FUNCTION_BLOCK fbMainStationProcess

VAR_INPUT
	(*fbStnSeqProcess*)
	bSavePB_Uni 									: BOOL; 														(*Universal*) (* Input - HMI - Save Push Button on Touchscreen*)
	bLoadPB_Uni 								: BOOL;														(*Universal*) (* Input - HMI - Load Push Button on Touchscreen*)
	bTrackerEn									: BOOL;														(*During Tracker, it will only call arm when process completed*)
	bTrackerBasedOnPreviousTime			: BOOL;

	(*fbGnrStationMasterController*)
	iCurrentStationAddress_Fix 					: INT;															(*Individual*) (* Input - Define current station no so that this fb know which array number to used*)
	iPreCallArmTime_Uni						: INT;															(*Universal*) (* Input - Pre-Call Arm Time, Program will call arm if the Total process timeEV Equal or Lesser than this value*)
	ARbAlternateStnEn : ARRAY [1..iAlternateSetQty] OF BOOL;
	AR2siAlternateStn : ARRAY [1..iAlternateSetQty, 1..iAlternateStnQty] OF INT;


END_VAR

VAR_IN_OUT PERSISTENT

	(*fbStnSeqProcess*)
(*	DsStnSeqProInput_Ind 						: DS_StnSeqProInput;											(*Individual*) (* Input - PV of Instrument (Temperature, pressure, vacuum and etc), Signal of Sensor to allowed program under the current station status.*)
*)	DSStnSeqProcessCtrl_Ind			 		: DS_fbStnSeqProcessCtrl;									(*Individual*) (* InOut - Link with fbStnSeqProcess, so that this fb know the full status of fbStnSeqProcess and determine which action to take*)

	DsStnSeqRepStore_Ind 						: DS_fbStationSequenceRecipeStore; 						(*Individual*) (* InOut - HMI - The full set of DataStructure-StationSequenceRecipe should selectively display on HMI so that user can customise the recipe by choosing/configure the parameters.*)
	DsStnSubRepStore_Ind 						: DS_fbStationSubRecipeStore; 								(*Individual*) (* InOut - HMI - The full set of DataStructure-StationSubRecipe should selectively display on HMI so that user can customise the recipe by choosing/configure the parameters.*)
	DsStnSeqRepCall_Ind 						: DS_fbStationSequenceRecipeCall;							(*Individual*) (* InOut - Used to call StationSequenceRecipe Detail from fbStationSequenceRecipe*)
	DsStnSubRepCall_Ind 						: DS_fbStationSubRecipeCall;								(*Individual*) (* InOut - Used to call StationSubRecipe Detail from fbStationSubRecipe*)

	(*fbGnrStationMasterController*)
	ARbProductRecipeCallEn_Uni 				: ARRAY [0..iStnQty] OF BOOL;					(*Universal*) (* Output - Link with fbGnrProductRecipeMemory, Array based on Current Station No, the fbGnrProductRecipeMemory will start Read info from Memory when this bool turn on*)
	ARiProductRecipeNoCall_Uni 				: ARRAY [0..iStnQty] OF INT;						(*Universal*) (* Output - Link with fbGnrProductRecipeMemory, Array based on Current Station No, the read out from fbGnrProductRecipeMemory is based on this Product Recipe No*)
	ARiProductRecipeStepCall_Uni 				: ARRAY [0..iStnQty] OF INT;						(*Universal*) (* Output - Link with fbGnrProductRecipeMemory, Array based on Current Station No, the read out from fbGnrProductRecipeMemory is based on this Product Recipe Step No*)

	DSfbGnrProductRecipeMemoryOut_Uni 		: DS_fbGnrProductRecipeMemoryOut;						(*Universal*) (* Input - Link with fbGnrProductRecipeMemory, all the read out info from fbGnrProductRecipeMemory will store in this DataStucture*)

	ARbArmReady_Uni							: ARRAY [1..iArmQty] OF BOOL;								(* Universal*) (* Input  - From ArmPnpFB, This signal is used to confirm if the arm is ready and idling*)

	ARiStnNoToCalledArm_Uni					: ARRAY [0..iArmQty] OF INT; 									(*Universal*) (* Output - Link with fbArmPnP, Array based on Arm No, The Int will store which Station that calling the Arm*)
	ARDSGnrFeedArmPnpParameter_Uni		: ARRAY [0..iArmQty] OF DSGnr_CalledArmPnpParameter; 	(*Universal*) (* Output - Link with fbArmPnP, Array based on Current Station No, Arm should move based on this DataStructure Info*)

	DSLdBasketInfo_Uni		 				: DS_BasketInfo;											(*Input - Loading CONFIRM Basket Info*)
	DSUldBasketInfo_Uni		 				: DS_BasketInfo;											(*Input - Uloading CONFIRM Basket Info*)
	ARDsStnBasketInfo_Uni					: ARRAY [1..iStnQty] OF DS_BasketInfo;						(*Input - Station Basket Info*)



END_VAR

VAR_OUTPUT PERSISTENT
	bSaveInd_Uni 								: BOOL; 														(*Universal*) (* Output - HMI - Save Indicator on Touchscreen*)
	bLoadInd_Uni 								: BOOL; 														(*Universal*) (* Output - HMI - Load Indicator on Touchscreen*)
(*	DSStnSeqProOutput_Ind 						:DS_StnSeqProOutput;										(*Individual*) (* Output - To Control Output - When process running, instrument should control by the output in this Data structure*)
*)
END_VAR



VAR PERSISTENT
	(*fbStnSeqProcess*)
	StnSeqProcessfb: fbStnSeqProcess;
	bStnSeqProcessStartInterlock			: BOOL;															(*Individual*) (* Input - Interlocking to Enable the StnSeqProcess Start Signal, It might used on those station with Sliding door for close confirmation before process start*)

	(*fbGnrStationMasterController*)
	GnrStationMasterControllerfb				: fbGnrStationMasterController;
	bStnSeqProcessSt						: BOOL;															(* Output - Link with fbStnSeqProcess, After Read out from fbGnrProductRecipeMemory, this fb will trigger this Bool to start the StnSeqProcess*)
	DSGnrBufferCalledArmPnpParameter 	: DSGnr_CalledArmPnpParameter;								(* Internal used, Buffer Data Structure read out from fbGnrProductRecipeMemory*)
	DSGnrBuffersPnpSequenceDescription	: STRING (99);														(* Internal used, Buffer Description read out from fbGnrProductRecipeMemory*)
	ARiPreviousStnSeqTotalProcessTime 	: ARRAY [0..iProductRecipeArrayQty] OF INT;					(* Internal used, Previous Total Process Time will save into this Array, Array based on StationSequenceNo*)
	iCallStep									: INT;																(* Internal used, to monitor the current Step so that you can indentify the error of this function block if stucked*)
	DSBasketInfo_Ind 							: DS_BasketInfo;												(*Individual*) (* InOut - Basket Information that comes into current station*)

END_VAR
VAR
	bLdStnConfirm: BOOL;
	bUldStnConfirm: BOOL;
	bStn1Confirm: BOOL;
	bGreaterStn1Confirm: BOOL;
	bLesserStnQtyConfirm: BOOL;
	bEqualStnQtyConfirm: BOOL;
	iTotalProcessTimeSV: INT;
END_VAR
VAR // added by the converter: edge detectors and wires of the graphical bodies
    _w1, _w2, _w3 : DS_BasketInfo;
END_VAR

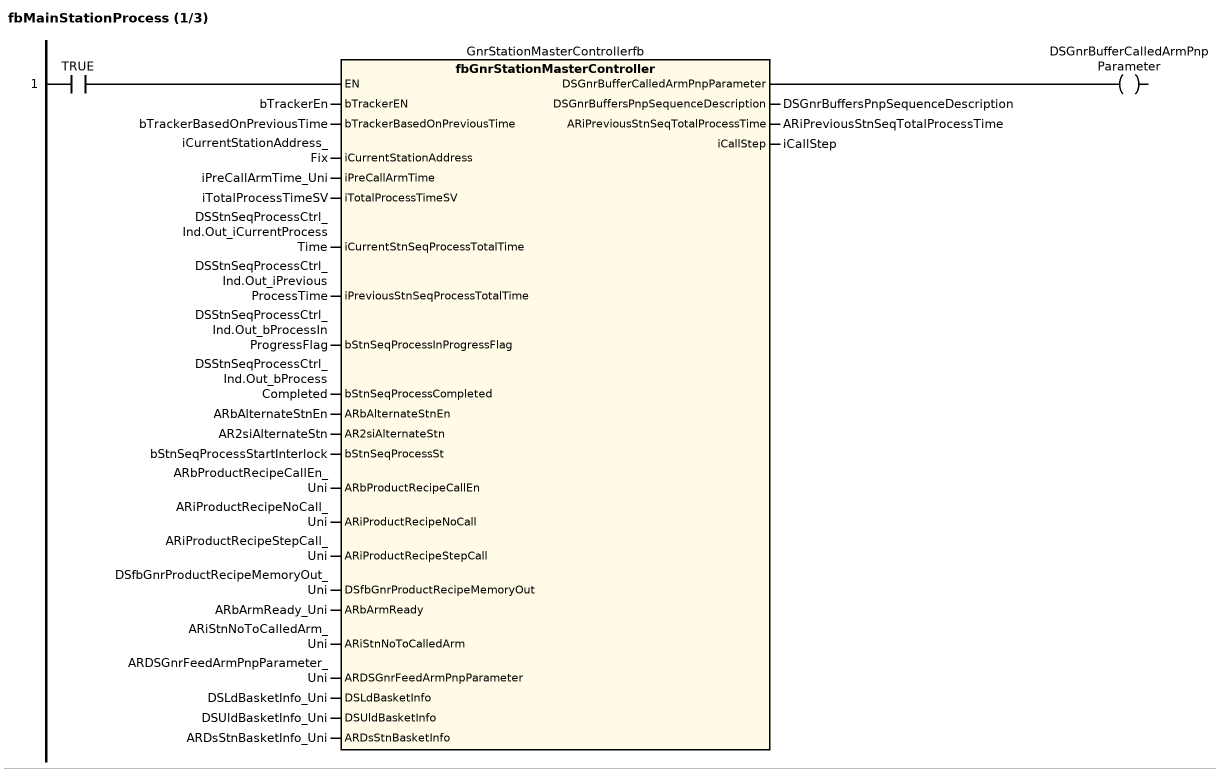
// NETWORK 1
GnrStationMasterControllerfb(
    bTrackerEN := bTrackerEn,
    bTrackerBasedOnPreviousTime := bTrackerBasedOnPreviousTime,
    iCurrentStationAddress := iCurrentStationAddress_Fix,
    iPreCallArmTime := iPreCallArmTime_Uni,
    iTotalProcessTimeSV := iTotalProcessTimeSV,
    iCurrentStnSeqProcessTotalTime := DSStnSeqProcessCtrl_Ind.Out_iCurrentProcessTime,
    iPreviousStnSeqProcessTotalTime := DSStnSeqProcessCtrl_Ind.Out_iPreviousProcessTime,
    bStnSeqProcessInProgressFlag := DSStnSeqProcessCtrl_Ind.Out_bProcessInProgressFlag,
    bStnSeqProcessCompleted := DSStnSeqProcessCtrl_Ind.Out_bProcessCompleted,
    ARbAlternateStnEn := ARbAlternateStnEn,
    AR2siAlternateStn := AR2siAlternateStn,
    bStnSeqProcessSt := bStnSeqProcessStartInterlock,
    ARbProductRecipeCallEn := ARbProductRecipeCallEn_Uni,
    ARiProductRecipeNoCall := ARiProductRecipeNoCall_Uni,
    ARiProductRecipeStepCall := ARiProductRecipeStepCall_Uni,
    DSfbGnrProductRecipeMemoryOut := DSfbGnrProductRecipeMemoryOut_Uni,
    ARbArmReady := ARbArmReady_Uni,
    ARiStnNoToCalledArm := ARiStnNoToCalledArm_Uni,
    ARDSGnrFeedArmPnpParameter := ARDSGnrFeedArmPnpParameter_Uni,
    DSLdBasketInfo := DSLdBasketInfo_Uni,
    DSUldBasketInfo := DSUldBasketInfo_Uni,
    ARDsStnBasketInfo := ARDsStnBasketInfo_Uni,
    DSGnrBuffersPnpSequenceDescription => DSGnrBuffersPnpSequenceDescription,
    ARiPreviousStnSeqTotalProcessTime => ARiPreviousStnSeqTotalProcessTime,
    iCallStep => iCallStep); // fbGnrStationMasterController
DSGnrBufferCalledArmPnpParameter := GnrStationMasterControllerfb.DSGnrBufferCalledArmPnpParameter;

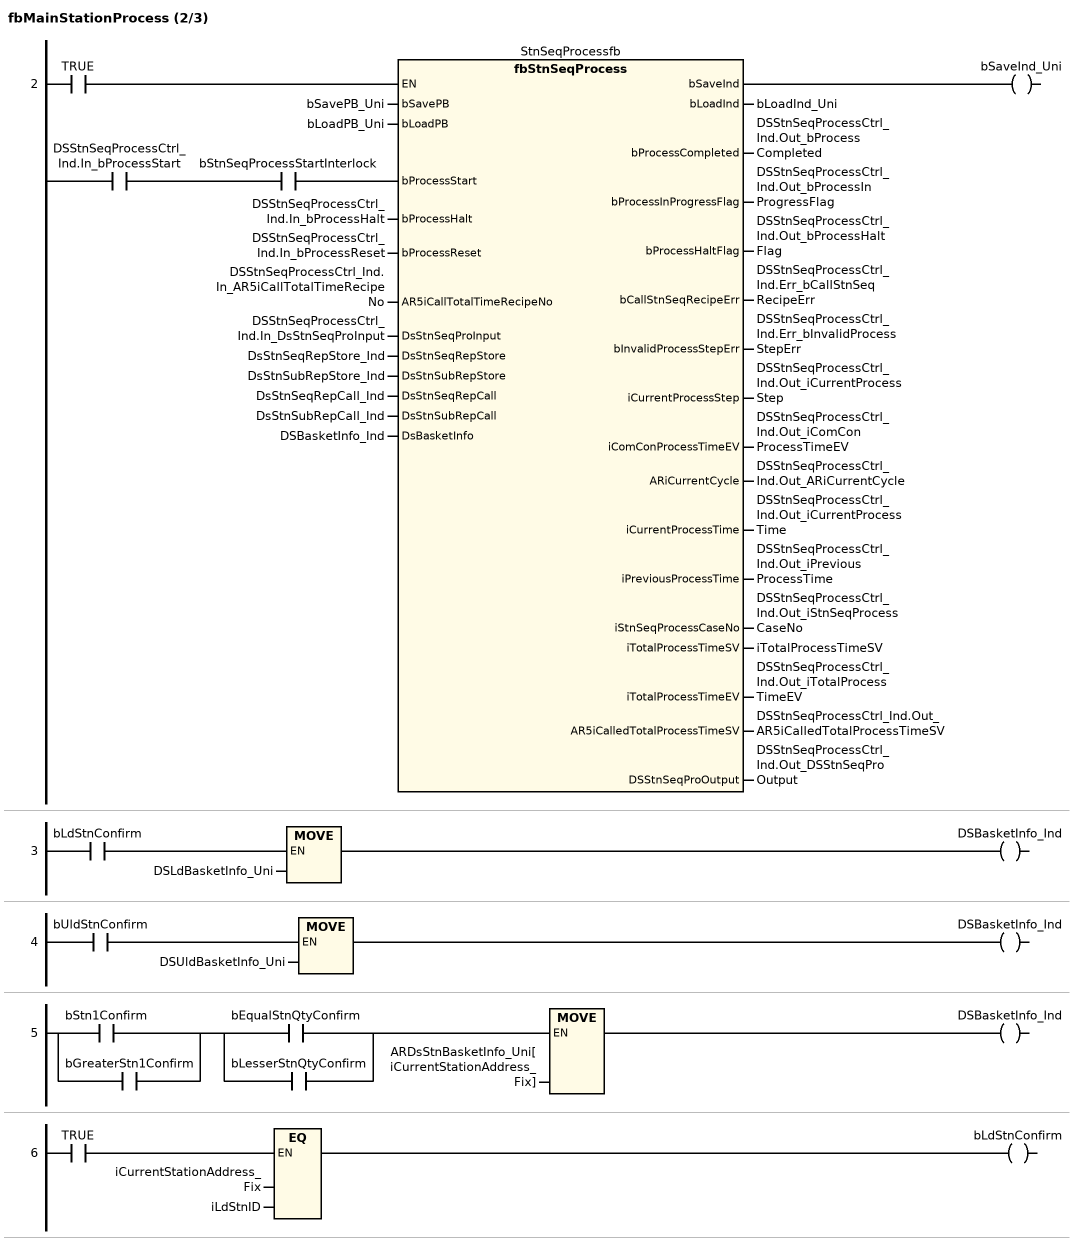
// NETWORK 2
StnSeqProcessfb(
    bSavePB := bSavePB_Uni,
    bLoadPB := bLoadPB_Uni,
    bProcessStart := DSStnSeqProcessCtrl_Ind.In_bProcessStart AND bStnSeqProcessStartInterlock,
    bProcessHalt := DSStnSeqProcessCtrl_Ind.In_bProcessHalt,
    bProcessReset := DSStnSeqProcessCtrl_Ind.In_bProcessReset,
    AR5iCallTotalTimeRecipeNo := DSStnSeqProcessCtrl_Ind.In_AR5iCallTotalTimeRecipeNo,
    DsStnSeqProInput := DSStnSeqProcessCtrl_Ind.In_DsStnSeqProInput,
    DsStnSeqRepStore := DsStnSeqRepStore_Ind,
    DsStnSubRepStore := DsStnSubRepStore_Ind,
    DsStnSeqRepCall := DsStnSeqRepCall_Ind,
    DsStnSubRepCall := DsStnSubRepCall_Ind,
    DsBasketInfo := DSBasketInfo_Ind,
    bLoadInd => bLoadInd_Uni,
    bProcessCompleted => DSStnSeqProcessCtrl_Ind.Out_bProcessCompleted,
    bProcessInProgressFlag => DSStnSeqProcessCtrl_Ind.Out_bProcessInProgressFlag,
    bProcessHaltFlag => DSStnSeqProcessCtrl_Ind.Out_bProcessHaltFlag,
    bCallStnSeqRecipeErr => DSStnSeqProcessCtrl_Ind.Err_bCallStnSeqRecipeErr,
    bInvalidProcessStepErr => DSStnSeqProcessCtrl_Ind.Err_bInvalidProcessStepErr,
    iCurrentProcessStep => DSStnSeqProcessCtrl_Ind.Out_iCurrentProcessStep,
    iComConProcessTimeEV => DSStnSeqProcessCtrl_Ind.Out_iComConProcessTimeEV,
    ARiCurrentCycle => DSStnSeqProcessCtrl_Ind.Out_ARiCurrentCycle,
    iCurrentProcessTime => DSStnSeqProcessCtrl_Ind.Out_iCurrentProcessTime,
    iPreviousProcessTime => DSStnSeqProcessCtrl_Ind.Out_iPreviousProcessTime,
    iStnSeqProcessCaseNo => DSStnSeqProcessCtrl_Ind.Out_iStnSeqProcessCaseNo,
    iTotalProcessTimeSV => iTotalProcessTimeSV,
    iTotalProcessTimeEV => DSStnSeqProcessCtrl_Ind.Out_iTotalProcessTimeEV,
    AR5iCalledTotalProcessTimeSV => DSStnSeqProcessCtrl_Ind.Out_AR5iCalledTotalProcessTimeSV,
    DSStnSeqProOutput => DSStnSeqProcessCtrl_Ind.Out_DSStnSeqProOutput); // fbStnSeqProcess
bSaveInd_Uni := StnSeqProcessfb.bSaveInd;

// NETWORK 3
IF bLdStnConfirm THEN _w1 := DSLdBasketInfo_Uni; END_IF
DSBasketInfo_Ind := _w1;

// NETWORK 4
IF bUldStnConfirm THEN _w2 := DSUldBasketInfo_Uni; END_IF
DSBasketInfo_Ind := _w2;

// NETWORK 5
IF (bStn1Confirm OR bGreaterStn1Confirm) AND (bEqualStnQtyConfirm OR bLesserStnQtyConfirm) THEN
    _w3 := ARDsStnBasketInfo_Uni[iCurrentStationAddress_Fix];
END_IF
DSBasketInfo_Ind := _w3;

// NETWORK 6
bLdStnConfirm := iCurrentStationAddress_Fix = iLdStnID;

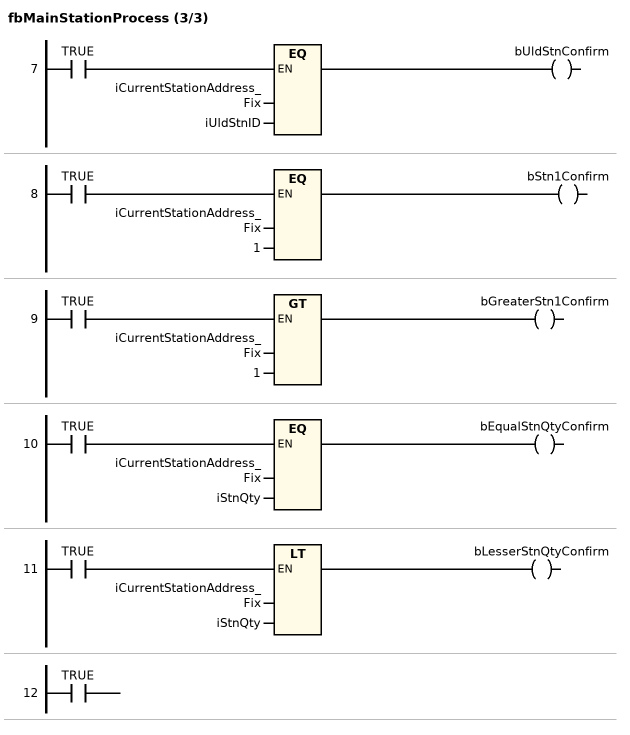
// NETWORK 7
bUldStnConfirm := iCurrentStationAddress_Fix = iUldStnID;

// NETWORK 8
bStn1Confirm := iCurrentStationAddress_Fix = 1;

// NETWORK 9
bGreaterStn1Confirm := iCurrentStationAddress_Fix > 1;

// NETWORK 10
bEqualStnQtyConfirm := iCurrentStationAddress_Fix = iStnQty;

// NETWORK 11
bLesserStnQtyConfirm := iCurrentStationAddress_Fix < iStnQty;

// NETWORK 12

END_FUNCTION_BLOCK

(* stored: Version 1.1.0.1, ProductVersion 3.1.4024.12
   POU fbMainStationProcess: Id {9432e160-822a-4b92-bbad-3371404532dd}, SpecialFunc None *)
